Staubli VAL3: onRun.pgx

public program onRun(string& x_sItem[])
  local num l_nValue
  local bool l_bCheck
  local num l_nIndex
  local num l_nOperator
  local string l_sName
begin
  // decompose
  call saveInOut:decompose_wait(x_sItem,l_sName,l_nOperator,l_nValue)
  if l_nIndex!=-1
    // check
    call condition(l_nOperator,l_nValue,l_sName,l_bCheck)
    // stop the robot
    if !l_bCheck
      call stopRobot()
      // <> >= > < <= ==
      do
        call condition(l_nOperator,l_nValue,l_sName,l_bCheck)
        delay(0)
      until l_bCheck==true
      // restart the robot
      cycleStatus:bWait=false
    endIf
  endIf
end
